{attribute addProperty BoxType "EL3423-0000-0016"}
{attribute addProperty Id "Total_StatusAT %I*Total_Status_F4CDE3E7144180Total_AdvancedAT %I*Total_Advanced_FCA492E91620Total_ActiveAT %I*Total_Active_10270F21192240Total_ApparentAT %I*Total_Apparent_A2159343192240Total_ReactiveAT %I*Total_Reactive_F843C78E192240Total_Statistic_PowerAT %I*Total_Statistic_Power_A2483F97288360Total_Statistic_PQFAT %I*Total_Statistic_PQF_4F621FA496120Total_Interval_EnergyAT %I*Total_Interval_Energy_3B88CECC296370IntervalAT %Q*Interval_ABCD96B2810WcStateAT %I*WcState_F855686C1620InfoDataAT %I*InfoData_BC63D37F80100"}
{attribute addProperty CRC "4178270661"}
{attribute addProperty SizeInBites "1520"}
{attribute addProperty SizeInBytes "190"}
TYPE EL3423_A72AC4D2 :
STRUCT
	{attribute addProperty Name "Total_Status"}
	Total_Status : Total_Status_F4CDE3E7;
	{attribute addProperty Name "Total_Advanced"}
	Total_Advanced : Total_Advanced_FCA492E9;
	{attribute addProperty Name "Total_Active"}
	Total_Active : Total_Active_10270F21;
	{attribute addProperty Name "Total_Apparent"}
	Total_Apparent : Total_Apparent_A2159343;
	{attribute addProperty Name "Total_Reactive"}
	Total_Reactive : Total_Reactive_F843C78E;
	{attribute addProperty Name "Total_Statistic_Power"}
	Total_Statistic_Power : Total_Statistic_Power_A2483F97;
	{attribute addProperty Name "Total_Statistic_PQF"}
	Total_Statistic_PQF : Total_Statistic_PQF_4F621FA4;
	{attribute addProperty Name "Total_Interval_Energy"}
	Total_Interval_Energy : Total_Interval_Energy_3B88CECC;
	{attribute addProperty Name "Interval"}
	Interval : Interval_ABCD96B2;
	{attribute addProperty Name "WcState"}
	WcState : WcState_F855686C;
	{attribute addProperty Name "InfoData"}
	InfoData : InfoData_BC63D37F;
END_STRUCT
END_TYPE

(* stored: Version 1.2.0.0, ProductVersion 3.1.4024.9
   DUT EL3423_A72AC4D2: Id {614284ac-0e8f-4aa2-97dd-89d3ebb249f6} *)
